FUNCTION_BLOCK FB_SUB_DT_TIME (* IEC 61131-3 DATE_AND_TIME - TIME *)
  (* Standard: IEC 61499-1 *)
  (* Version 0.0, 2006-09-11, JHC, Holobloc Inc *)
  (* Compiler header: package fb.rt.math; *)
  (* Compiler Java Sun JDK 1.5.0 *)
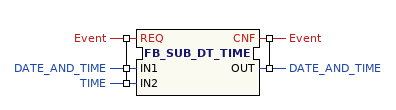
  EVENT_INPUT
    REQ WITH IN1, IN2;
  END_EVENT
  EVENT_OUTPUT
    CNF WITH OUT;
  END_EVENT
  VAR_INPUT
    IN1 : DATE_AND_TIME; (* Augend *)
    IN2 : TIME; (* Addend *)
  END_VAR
  VAR_OUTPUT
    OUT : DATE_AND_TIME; (* Sum *)
  END_VAR
END_FUNCTION_BLOCK
